// TIA Portal V17 export
// export: Created 2024-08-09T12:50:43.6499454Z, ExportSetting WithDefaults, DisplayName Totally Integrated Automation Portal, DisplayVersion V17 Update 7, DisplayName TIA Portal Openness, DisplayVersion V17 Update 7, DisplayName TIA Portal Version Control Interface, DisplayVersion V17, DisplayName STEP 7 Professional, DisplayVersion V17 Update 7, DisplayName STEP 7 Safety, DisplayVersion V17 Update 6, DisplayName WinCC Professional, DisplayVersion V17 Update 7
DATA_BLOCK "DB_EXECUTE_StoredProcedure"   // DB28
VERSION : 0.1
// stored: AutoNumber true, DBAccessibleFromOPCUA true, DBAccessibleFromWebserver true, InstanceOfName FB_EXECUTE_StoredProcedure, InstanceOfType FB
"FB_EXECUTE_StoredProcedure"
   // VAR_INPUT
   //    procedure_name : String;
   //    values_of_record : Array[0..20] of String;
   //    parameters_number : SInt;
   // END_VAR
   // VAR_OUTPUT
   //    xReady : Bool;
   //    xBusy : Bool;
   //    xDone : Bool;
   //    xError : Bool;
   //    diResultState : DInt;
   //    sResult : WString[6000];
   // END_VAR
   // VAR_IN_OUT
   //    stSql4SiemensInterface : "utSql4SiemensInterface";
   //    xExecute : Bool;
   // END_VAR
   // VAR
   //    iStep : Int;
   //    diDoneCount : DInt;
   //    diErrorCount : DInt;
   // END_VAR
   // VAR RETAIN
   //    query_assembled : String;
   // END_VAR
BEGIN
END_DATA_BLOCK
